// TIA Portal V17 export
// export: Created 2025-03-10T12:18:00.3479262Z, ExportSetting WithDefaults, DisplayName Totally Integrated Automation Portal, DisplayVersion V17 Update 8, DisplayName TIA Portal Openness, DisplayVersion V17 Update 8, DisplayName TIA Portal Version Control Interface, DisplayVersion V17, DisplayName SINAMICS Startdrive Advanced, DisplayVersion V17 SP2, DisplayName SINAMICS Startdrive G110M, G120, G120C, G120D, G120P, G115D, DisplayVersion V17 SP2, DisplayName SINAMICS Startdrive G130, G150, S120, S150, SINAMICS MV, S210, DisplayVersion V17 SP2, DisplayName STEP 7 Professional, DisplayVersion V17 Update 8, DisplayName SINUMERIK ONE STEP 7 Toolbox, DisplayVersion V17 Update 12, DisplayName SINUMERIK 840D sl STEP 7 Toolbox, DisplayVersion V17 Update 12, DisplayName STEP 7 Safety, DisplayVersion V17 Update 6, DisplayName WinCC Advanced, DisplayVersion V17 Update 8
TYPE "MPP_OUTPUTS"
// stored: IsFailsafeCompliant false
   STRUCT
      O_HS1 : Bool;   // MPP483 LAMP - CONTROL ON / LAMP - CONTROL ON
      O_HS2 : Bool;   // MPP483 LAMP - START / LAMP - START
      O_HS3 : Bool;   // MPP483 LAMP - HOME / LAMP - HOME
      O_HS4 : Bool;   // MPP483 LAMP - RESET FAULT / LAMP - RESET FAULT
      O_HS14 : Bool;   // MPP483 LAMP - / LAMP -
      O_HS15 : Bool;   // MPP483 LAMP - / LAMP -
      O_HS7 : Bool;   // MPP483 LAMP - CONTROL OFF / LAMP - CONTROL OFF
      O_HS8 : Bool;   // MPP483 LAMP - STOP END OF CYCLE / LAMP - STOP END OF CYCLE
      O_HS9 : Bool;   // MPP483 LAMP - IMMEDIATE STOP / LAMP - IMMEDIATE STOP
      O_HS10 : Bool;   // MPP483 LAMP - SAFETY DOOR CLOSED & LOCKED / LAMP - SAFETY DOOR CLOSED AND LOCKED
      O_1_2 : Bool;   // NOT USED
      O_1_3 : Bool;   // NOT USED
      O_1_4 : Bool;   // NOT USED
      O_1_5 : Bool;   // NOT USED
      O_1_6 : Bool;   // NOT USED
      O_1_7 : Bool;   // NOT USED
      O_H51 : Bool;   // H51 EXTENSION KEY - / H51 - EXTENSION KEY
      O_H52 : Bool;   // H52 EXTENSION KEY - / H52 - EXTENSION KEY
      O_H53 : Bool;   // H53 EXTENSION KEY - / H53 - EXTENSION KEY
      O_H54 : Bool;   // H54 EXTENSION KEY - / H54 - EXTENSION KEY
      O_H55 : Bool;   // H55 EXTENSION KEY - / H55 - EXTENSION KEY
      O_H56 : Bool;   // H56 EXTENSION KEY - / H56 - EXTENSION KEY
      O_H57 : Bool;   // H57 EXTENSION KEY - / H57 - EXTENSION KEY
      O_H58 : Bool;   // H58 EXTENSION KEY - / H58 - EXTENSION KEY
      O_H59 : Bool;   // H59 EXTENSION KEY - / H59 - EXTENSION KEY
      O_H60 : Bool;   // H60 EXTENSION KEY - / H60 - EXTENSION KEY
      O_HS13 : Bool;   // HS13 - FEEDBACK EMERGENCY STOP
      O_H61_SR_PUSH_BUTTON : Bool;   // H61 - SR KEY / H61 - SR PUSH BUTTON
      O_3_4 : Bool;   // NOT USED
      O_3_5 : Bool;   // NOT USED
      O_3_6 : Bool;   // NOT USED
      O_3_7 : Bool;   // NOT USED
      O_HF1 : Bool;   // MPP483 LAMP - CONTINUOUS CYCLE / LAMP - CONTINUOUS CYCLE
      O_HF2 : Bool;   // MPP483 LAMP - AUTOMATIC MODE / LAMP - AUTOMATIC MODE
      O_HF3 : Bool;   // MPP483 LAMP - SINGLE BLOCK / LAMP - SINGLE BLOCK
      O_HF4 : Bool;   // MPP483 LAMP - NC STOP / LAMP - NC STOP
      O_HF5 : Bool;   // MPP483 LAMP - NC START / LAMP - NC START
      O_HF6 : Bool;   // MPP483 LAMP - ONE CYCLE / LAMP - SINGLE CYCLE
      O_HF7 : Bool;   // MPP483 LAMP - MDA MODE / LAMP - MDA MODE
      O_HF8 : Bool;   // MPP483 LAMP - NEXT AXES / LAMP - NEXT AXES
      O_HF9 : Bool;   // MPP483 LAMP - FEEDRATE STOP / LAMP - FEEDRATE STOP
      O_HF10 : Bool;   // MPP483 LAMP - FEEDRATE START / LAMP - FEEDRATE START
      O_HF11 : Bool;   // MPP483 LAMP - STEP BY STEP CYCLE / LAMP - STEP BY STEP CYCLE
      O_HF12 : Bool;   // MPP483 LAMP - JOG MODE / LAMP - JOG MODE
      O_HF13 : Bool;   // MPP483 LAMP - (X1 - W) AXES / LAMP - (X1 - W) AXES
      O_HF14 : Bool;   // MPP483 LAMP - (Y1 - E) AXES / LAMP - (Y1 - E) AXES
      O_HF15 : Bool;   // MPP483 LAMP - Z11 AXIS / LAMP - Z11 AXIS
      O_HF16 : Bool;   // MPP483 LAMP - SETUP MODE / LAMP - SETUP MODE
      O_HF17 : Bool;   // MPP483 LAMP - REFERENCE POINT MODE / LAMP - REFERENCE POINT MODE
      O_HF18 : Bool;   // MPP483 LAMP - (A - U1 - C) AXES / LAMP - (A - U1 - C) AXES
      O_HF19 : Bool;   // MPP483 LAMP - B AXIS / LAMP - B AXIS
      O_HF20 : Bool;   // MPP483 LAMP - (Q1 - Z12) AXES / LAMP - (Q1 - Z12) AXES
      O_HF21 : Bool;   // MPP483 LAMP - RESET / LAMP - RESET
      O_HF22 : Bool;   // MPP483 LAMP - INCREMENTAL MODE / LAMP - INCREMENTAL MODE
      O_HF23 : Bool;   // MPP483 LAMP - MINUS DIRECTION / LAMP - MINUS DIRECTION
      O_HF24 : Bool;   // MPP483 LAMP - RAPID / LAMP - RAPID
      O_HF25 : Bool;   // MPP483 LAMP - PLUS DIRECTION / LAMP - PLUS DIRECTION
      O_7_1 : Bool;   // NOT USED
      O_7_2 : Bool;   // NOT USED
      O_7_3 : Bool;   // NOT USED
      O_7_4 : Bool;   // NOT USED
      O_7_5 : Bool;   // NOT USED
      O_7_6 : Bool;   // NOT USED
      O_7_7 : Bool;   // NOT USED
   END_STRUCT;
END_TYPE
